Staubli VAL3: motionControl.pgx

public program motionControl()
  local MotionCmd l_mTrajPt
  local bool l_bFlag
  local MotionCmd l_motion
  local num l_nTime
  local bool l_bStopAndClean
  local num l_nElems
begin
  // Copyright (c) 2016, Ocado Technology - Robotics Research Team
  //
  // Licensed under the Apache License, Version 2.0 (the "License");
  // you may not use this file except in compliance with the License.
  // You may obtain a copy of the License at
  //
  //     http://www.apache.org/licenses/LICENSE-2.0
  //
  // Unless required by applicable law or agreed to in writing, software
  // distributed under the License is distributed on an "AS IS" BASIS,
  // WITHOUT WARRANTIES OR CONDITIONS OF ANY KIND, either express or implied.
  // See the License for the specific language governing permissions and
  // limitations under the License.



  nMoveId = -1

  while (true)
    // check connection status, and whether to stop motion
    if (nInConnFlag == 1 and nOutConnFlag == 1 and bStopNow == false)

      // process trajectory point from trajectory buffer
      call libQueueFuncs:getNumElems(qTrajPtBuffer, l_nElems)
      if (l_nElems > 0)
        call libQueueFuncs:pop(qTrajPtBuffer,l_mTrajPt, l_bFlag)
        if (l_bFlag == true)
          nPtsPopped = nPtsPopped + 1
          call libQueueFuncs:push(qMoveBuffer,l_mTrajPt,l_bFlag)
        endIf
      endIf

      // process motion command from move buffer
      // @TODO move buffer should have elements previously interpolated to ensure they are 4 ms apart
      call libQueueFuncs:getNumElems(qMoveBuffer, l_nElems)
      if (l_nElems > 0)
        call libQueueFuncs:pop(qMoveBuffer,l_motion,l_bFlag)
        if (l_bFlag == true)
          nMovePts = nMovePts + 1
          // contrary to what we did earlier, we unconditionally add the traj pt to the motion queue:
          // there doesn't appear to be a way to compare the 'current pose' of the robot to the pts
          // in the trajectory at the appropriate time (ie: when the robot is in motion and about to
          // start executing the segment towards 'l_motion').
          // Checking for dist(l_motion, herej()) (pseudo code) would not be correct as there will
          // always be a delay in the data coming out of herej() and the actual pose of the robot.
          // @TODO potentially set move id according to sequence value
          nMoveId = movej(l_motion.jJointRx, tTool, l_motion.mDesc)
        endIf
      endIf
    else
      // stop immediately -- resetMotion() also resets moveId
      resetMotion()
      // clear buffers
      call libQueueFuncs:clear(qTrajPtBuffer)
      call libQueueFuncs:clear(qMoveBuffer)
      bStopNow = false

      // debug
      nPtsPopped = 0
      nMovePts = 0
    endIf

    nMotionProgress = getMoveId()

    // sequence task
    delay(0)
  endWhile
end
